(* CODESYS project 信号機_駅制御_柴山.project

Project tree, tasks and I/O mapping:
  Device : CODESYS Control Win V3 x64, 3S - Smart Software Solutions GmbH, version 3.5.11.40
    application Application
      libraries: Standard, * (System); File Access, 3.5.7.0 (3S - Smart Software Solutions GmbH); Network, 3.5.7.0 (3S - Smart Software Solutions GmbH)
      task MainTask (cyclic, interval 4 ms, priority 0) calls EtherCAT_Master.EtherCAT_Task [EtherCAT_Master.EtherCAT_Task], StationControlMain
      program StationControlMain [ST]
      function block OnOffDelay [ST]
      function block TrainDetection [ST]
      SignalControl/
        function block FourStateSignal [ST]
        function block FourStateSignalDecoder [ST]
        function block ThreeStateSignal [ST]
        function block ThreeStateSignalDecoder [ST]
        function block FourStateWarningSignalDecoder [ST]
      declarations NVL_StationControl
      global variables NVL_StationStatus
      global variables ControlLever
      function block SwitchControl [ST]
      function block SignalControl [ST]
      Encode/
        function block Encode_Status [ST]
        function EncodeSignalStatusOne [ST]
        function EncodeDetectionOne [ST]
        function EncodeSignalLockStatusOne [ST]
        function EncodeSwitchStatusOne [ST]
        function EncodeSwitchLockStatusOne [ST]
        function EncodeRouteStatusOne [ST]
      Decode/
        function DecodeSwitchLeverOne [ST]
        function block Decode_Levers [ST]
        function DecodeSignalLeverOne [ST]
      function block RouteControl [ST]
    EtherCAT_Master : EtherCAT Master, 3S - Smart Software Solutions GmbH, version 3.5.11.40
        settings: NetworkName = 'イーサネット'; NetworkName = "イーサネット"; SrcAddress1 = 60449; SrcAddress2 = 3851182877
      NX_ECC202 : NX-ECC202 EtherCAT coupler V1.2, OMRON Corporation, order no. NX-ECC202, version Revision=16#00010002
          settings: ModularDevice = True; Number of Outputs = 0; Number of Infos about Outputs = 0; MDP_InputOffsets = [0,0,0,0,272]; MDP_OutputOffsets = [0,0,32,64,0]; StationAlias = 0; Sync.Length = 12; Sync.Length = 38; FMMU.Length = 12; FMMU.Length = 38; Number of RxPDOs of the Slave = 3; Number of TxPDOs of the Slave = 4; DC sync0 cycletime = 4000; DC sync1 cycletime = 4000; Number of SDO = 1; RxTxPdo.NumberofExcludes = 0; RxTxPdo.NumberofEntries = 1; RxTxPdo.Index = 16#1600; RxTxPdo.Fixed = True; RxTxPdo.Mandatory = True; RxTxPdo.Virtual = False; RxTxPdo.Sm = 2; RxTxPdo.Su = 0; RxTxPdo.Name = 'Output Data Set 1'; RxTxPdo.DependOnSlot = True; RxTxPdo.DependOnSlotGroup = False; RxTxPdo.OverwrittenByModule = True; Output Bit 32 bits.Index = 16#7003; Output Bit 32 bits.SubIndex = 1; Output Bit 32 bits.Size = 32; Output Bit 32 bits.Offset = 0; Output Bit 32 bits.DependOnSlot = True; Output Bit 32 bits.DependOnSlotGroup = True; RxTxPdo.NumberofExcludes = 0; RxTxPdo.NumberofEntries = 1; RxTxPdo.Index = 16#1604; RxTxPdo.Fixed = True; RxTxPdo.Mandatory = True; RxTxPdo.Virtual = False; RxTxPdo.Sm = 2;
            RxTxPdo.Su = 0; RxTxPdo.Name = 'Output Data Set 1'; RxTxPdo.DependOnSlot = True; RxTxPdo.DependOnSlotGroup = False; RxTxPdo.OverwrittenByModule = True; Output Bit 32 bits.Index = 16#7023; Output Bit 32 bits.SubIndex = 1; Output Bit 32 bits.Size = 32; Output Bit 32 bits.Offset = 0; Output Bit 32 bits.DependOnSlot = True; Output Bit 32 bits.DependOnSlotGroup = True; RxTxPdo.NumberofExcludes = 0; RxTxPdo.NumberofEntries = 1; RxTxPdo.Index = 16#1608; RxTxPdo.Fixed = True; RxTxPdo.Mandatory = True; RxTxPdo.Virtual = False; RxTxPdo.Sm = 2; RxTxPdo.Su = 0; RxTxPdo.Name = 'Output Data Set 1'; RxTxPdo.DependOnSlot = True; RxTxPdo.DependOnSlotGroup = False; RxTxPdo.OverwrittenByModule = True; Output Bit 32 bits.Index = 16#7043; Output Bit 32 bits.SubIndex = 1; Output Bit 32 bits.Size = 32; Output Bit 32 bits.Offset = 0; Output Bit 32 bits.DependOnSlot = True; Output Bit 32 bits.DependOnSlotGroup = True; RxTxPdo.NumberofExcludes = 0; RxTxPdo.NumberofEntries = 2; RxTxPdo.Index = 16#1BF8; RxTxPdo.Fixed = False; RxTxPdo.Mandatory = False; RxTxPdo.Virtual = False; RxTxPdo.Sm = 3; RxTxPdo.Su = 3; RxTxPdo.Name = '505th transmit PDO Mapping'; RxTxPdo.DependOnSlot = False; RxTxPdo.DependOnSlotGroup = False;
            RxTxPdo.OverwrittenByModule = False; NX Unit Registration Status 125.Index = 16#3003; NX Unit Registration Status 125.SubIndex = 4; NX Unit Registration Status 125.Size = 128; NX Unit Registration Status 125.Offset = 0; NX Unit Registration Status 125.DependOnSlot = False; NX Unit Registration Status 125.DependOnSlotGroup = False; NX Unit I/O Data Active Status 125.Index = 16#3006; NX Unit I/O Data Active Status 125.SubIndex = 4; NX Unit I/O Data Active Status 125.Size = 128; NX Unit I/O Data Active Status 125.Offset = 0; NX Unit I/O Data Active Status 125.DependOnSlot = False; NX Unit I/O Data Active Status 125.DependOnSlotGroup = False; RxTxPdo.NumberofExcludes = 0; RxTxPdo.NumberofEntries = 1; RxTxPdo.Index = 16#1BFF; RxTxPdo.Fixed = True; RxTxPdo.Mandatory = False; RxTxPdo.Virtual = False; RxTxPdo.Sm = 3; RxTxPdo.Su = 3; RxTxPdo.Name = '512th transmit PDO Mapping'; RxTxPdo.DependOnSlot = False; RxTxPdo.DependOnSlotGroup = False; RxTxPdo.OverwrittenByModule = False; Sysmac Error Status.Index = 16#2002; Sysmac Error Status.SubIndex = 1; Sysmac Error Status.Size = 8; Sysmac Error Status.Offset = 0; Sysmac Error Status.DependOnSlot = False; Sysmac Error Status.DependOnSlotGroup = False; RxTxPdo.NumberofExcludes = 0; RxTxPdo.NumberofEntries = 1; RxTxPdo.Index = 16#1BF4; RxTxPdo.Fixed = True; RxTxPdo.Mandatory = False; RxTxPdo.Virtual = False; RxTxPdo.Sm = 3; RxTxPdo.Su = 3; RxTxPdo.Name = '501st transmit PDO Mapping';
            RxTxPdo.DependOnSlot = False; RxTxPdo.DependOnSlotGroup = False; RxTxPdo.OverwrittenByModule = False; Entry.Offset = 0; Entry.DependOnSlot = False; Entry.DependOnSlotGroup = False; RxTxPdo.NumberofExcludes = 0; RxTxPdo.NumberofEntries = 1; RxTxPdo.Index = 16#1A0C; RxTxPdo.Fixed = True; RxTxPdo.Mandatory = True; RxTxPdo.Virtual = False; RxTxPdo.Sm = 3; RxTxPdo.Su = 0; RxTxPdo.Name = 'Input Data Set  1'; RxTxPdo.DependOnSlot = True; RxTxPdo.DependOnSlotGroup = False; RxTxPdo.OverwrittenByModule = True; Input Bit 32 bits.Index = 16#6063; Input Bit 32 bits.SubIndex = 1; Input Bit 32 bits.Size = 32; Input Bit 32 bits.Offset = 0; Input Bit 32 bits.DependOnSlot = True; Input Bit 32 bits.DependOnSlotGroup = True; Output Bit 32 bits.Name = 'Output Bit 32 bits'; Output Bit 32 bits.DataType = 'UDINT'; Output Bit 32 bits.Default = ''; Output Bit 32 bits.Comment = ''; Output Bit 32 bits.Name = 'Output Bit 32 bits'; Output Bit 32 bits.DataType = 'UDINT'; Output Bit 32 bits.Default = ''; Output Bit 32 bits.Comment = ''; Output Bit 32 bits.Name = 'Output Bit 32 bits'; Output Bit 32 bits.DataType = 'UDINT'; Output Bit 32 bits.Default = ''; Output Bit 32 bits.Comment = ''; NX Unit Registration Status 125.Name = 'NX Unit Registration Status 125'; NX Unit Registration Status 125.DataType = 'ARRAY [0..15] OF BYTE'; NX Unit Registration Status 125.Default = ''; NX Unit Registration Status 125.Comment = '';
            NX Unit I/O Data Active Status 125.Name = 'NX Unit I/O Data Active Status 125'; NX Unit I/O Data Active Status 125.DataType = 'ARRAY [0..15] OF BYTE'; NX Unit I/O Data Active Status 125.Default = ''; NX Unit I/O Data Active Status 125.Comment = ''; Sysmac Error Status.Name = 'Sysmac Error Status'; Sysmac Error Status.DataType = 'USINT'; Sysmac Error Status.Default = ''; Sysmac Error Status.Comment = ''; Entry.Default = ''; Input Bit 32 bits.Name = 'Input Bit 32 bits'; Input Bit 32 bits.DataType = 'UDINT'; Input Bit 32 bits.Default = ''; Input Bit 32 bits.Comment = ''
          unmapped channels: NX Unit Registration Status 125, NX Unit I/O Data Active Status 125, Sysmac Error Status, 
        NX_OD6121_5 : General output, OMRON Corporation, order no. NX-OD6121-5, version 0
            settings: Number of Outputs = 1; Number of Infos about Outputs = 1; Output Bit 32 bits.Offset = 0; Output Bit 32 bits.DependOnSlot = True; Output Bit 32 bits.DependOnSlotGroup = True; Output Bit 32 bits.Default = ''
            unmapped channels: Output Bit 32 bits
        NX_ID6142_5_1 : General input, OMRON Corporation, order no. NX-ID6142-5, version 0
            settings: Number of Inputs = 1; Number of Infos about Inputs = 1; Input Bit 32 bits.Index = 16#6063; Input Bit 32 bits.SubIndex = 1; Input Bit 32 bits.Size = 32; Input Bit 32 bits.Offset = 0; Input Bit 32 bits.DependOnSlot = True; Input Bit 32 bits.DependOnSlotGroup = True; Input Bit 32 bits.Name = 'Input Bit 32 bits'; Input Bit 32 bits.DataType = 'UDINT'; Input Bit 32 bits.Default = ''; Input Bit 32 bits.Comment = ''
            unmapped channels: Input Bit 32 bits
        NX_OD6121_5_2 : General output, OMRON Corporation, order no. NX-OD6121-5, version 0
            settings: Number of Outputs = 1; Number of Infos about Outputs = 1; Output Bit 32 bits.Index = 16#7043; Output Bit 32 bits.SubIndex = 1; Output Bit 32 bits.Size = 32; Output Bit 32 bits.Offset = 0; Output Bit 32 bits.DependOnSlot = True; Output Bit 32 bits.DependOnSlotGroup = True; Output Bit 32 bits.Name = 'Output Bit 32 bits'; Output Bit 32 bits.DataType = 'UDINT'; Output Bit 32 bits.Default = ''; Output Bit 32 bits.Comment = ''
            unmapped channels: Output Bit 32 bits
        NX_OD6121_5_1 : General output, OMRON Corporation, order no. NX-OD6121-5, version 0
            settings: Number of Outputs = 1; Number of Infos about Outputs = 1; Output Bit 32 bits.Index = 16#7023; Output Bit 32 bits.SubIndex = 1; Output Bit 32 bits.Size = 32; Output Bit 32 bits.Offset = 0; Output Bit 32 bits.DependOnSlot = True; Output Bit 32 bits.DependOnSlotGroup = True; Output Bit 32 bits.Name = 'Output Bit 32 bits'; Output Bit 32 bits.DataType = 'UDINT'; Output Bit 32 bits.Default = ''; Output Bit 32 bits.Comment = ''
            unmapped channels: Output Bit 32 bits
  data type E_SIGNAL_STATUS
*)

// E_SIGNAL_STATUS
TYPE E_SIGNAL_STATUS :
(
	R_Stop, YY_Warnig, Y_Caution, YG_Slowdown, G_Go
);
END_TYPE

// Device/Application/NVL_StationControl
//このグローバル変数リストはネットワーク経由受信です。
//送信者: ファイル 'C:\Users\Tomonobu\Documents\home\CodesysProject\StationControl.gvl' からインポートされました
//プロトコル: UDP

{attribute 'qualified_only'}
VAR_GLOBAL
	singal_lever_status: ARRAY[0..15] OF UINT;
	switch_lever_nml: ARRAY[0..15] OF UINT;
	switch_lever_rev: ARRAY[0..15] OF UINT;
END_VAR

// Device/Application/NVL_StationStatus
{attribute 'qualified_only'}
VAR_GLOBAL
	signal_display: ARRAY[0..15] OF E_SIGNAL_STATUS;
	signal_satus: ARRAY[0..15] OF UINT;
	signal_locked: ARRAY[0..15] OF UINT;
	singal_reserve0: ARRAY[0..15] OF UINT;
	switch_status: ARRAY[0..15] OF UINT;
	switch_locked: ARRAY[0..15] OF UINT;
	switch_reserve0: ARRAY[0..15] OF UINT;
	section_status: ARRAY[0..15] OF UINT;
END_VAR

// Device/Application/ControlLever
{attribute 'qualified_only'}
VAR_GLOBAL
	Switch_31Nml: BOOL;
	Switch_21Nml: BOOL;
	Switch_31Rev: BOOL;
	Switch_21Rev: BOOL;
	Route_11Nml: BOOL;
	Route_11Rev: BOOL;
	Route_12Nml: BOOL;
	Route_12Rev: BOOL;
	Signal_2R: BOOL;
	Signal_3R: BOOL;
	Signal_4R: BOOL;
	Signal_5R: BOOL;
	Signal_2L: BOOL;
	Signal_3L: BOOL;
	Signal_4L: BOOL;
	Signal_5L: BOOL;
END_VAR

// Device/Application/StationControlMain
PROGRAM StationControlMain
VAR
	Detect_Sensor : TrainDetection; 
	Input_Decode  : Decode_Levers;
	Output_Encode : Encode_Status;
	abDetectInfo_All : ARRAY[0..15] OF BOOL;

	Signal_2R: SignalControl;
	Signal_3R: SignalControl;

	Signal_2L: SignalControl;
	Signal_3L: SignalControl;

	Route_11: RouteControl;
	Route_12: RouteControl;
	
	Switch_31: SwitchControl;
	Switch_21: SwitchControl;

	Signal_2L_Decode: FourStateWarningSignalDecoder;
	Signal_3L_Decode: ThreeStateSignalDecoder;
	Signal_2R_Decode: ThreeStateSignalDecoder;
 	Signal_3R_Decode: FourStateWarningSignalDecoder;
	
	// 在線検知
	bExist_31T: BOOL;
	bExist_21T: BOOL;
	bExist_2RT: BOOL;
	bExist_5RT: BOOL;
	
END_VAR

Input_Decode();
Output_Encode(sig_2R:=Signal_2R, sig_3R:=Signal_3R,
	          sig_2L:=Signal_2L, sig_3L:=Signal_3L,
			  swt_31:=Switch_31, swt_21:=Switch_21, 
			  route_11:=Route_11, route_12:=Route_12,
              abDetect:=abDetectInfo_All);
Detect_Sensor(abDetect => abDetectInfo_All);

// 在線検知信号
bExist_31T := abDetectInfo_All[0];
bExist_21T := abDetectInfo_All[1];
bExist_2RT := abDetectInfo_All[2];
bExist_5RT := abDetectInfo_All[3];

// 鎖錠信号
// 2L
IF NOT Switch_21.bStatusNormal THEN
	Signal_2L.bLockedNml := TRUE;
ELSE
	Signal_2L.bLockedNml := FALSE; 
END_IF
Signal_2L.bLockedRev := FALSE;

Signal_2L.bRouteAcquired := NOT Switch_31.bStatusNormal;

// 3L
IF Switch_31.bStatusNormal THEN
	Signal_3L.bLockedNml := TRUE;
ELSE
	SIgnal_3L.bLockedNml := FALSE;
END_IF

IF (Signal_2L.bLockActive AND NOT Signal_3L.bStatusNormal) THEN
	Signal_3L.bLockedRev := TRUE;
ELSE 
	Signal_3L.bLockedRev := FALSE;
END_IF

// 2R
IF Switch_21.bStatusNormal THEN
	Signal_2R.bLockedNml := TRUE;
ELSE
	Signal_2R.bLockedNml := FALSE;
END_IF

IF (Signal_3R.bLockActive AND NOT Signal_2R.bStatusNormal) THEN
	Signal_2R.bLockedRev := TRUE;
ELSE 
	Signal_2R.bLockedRev := FALSE;
END_IF

//5R
IF NOT Switch_31.bStatusNormal THEN
	Signal_3R.bLockedNml := TRUE;
ELSE
	Signal_3R.bLockedNml := FALSE;
END_IF
Signal_3R.bLockedRev := FALSE;

Signal_3R.bRouteAcquired := NOT Switch_21.bStatusNormal;

// 31
IF Signal_3R.bLockActive THEN
	Switch_31.bLockedNml := TRUE;
ELSE
	Switch_31.bLockedNml := FALSE;
END_IF

IF Signal_3L.bLockActive OR
	(Route_12.bLockActive AND NOT Switch_31.bStatusNormal) THEN
	Switch_31.bLockedRev := TRUE;
ELSE
	Switch_31.bLockedRev := FALSE;
END_IF

// 21
IF Signal_2L.bLockActive THEN
	Switch_21.bLockedNml := TRUE;
ELSE
	Switch_21.bLockedNml := FALSE;
END_IF

IF Signal_2R.bLockActive OR
	(Route_11.bLockActive AND NOT Switch_21.bStatusNormal) THEN
	Switch_21.bLockedRev := TRUE;
ELSE
	Switch_21.bLockedRev := FALSE;
END_IF

// 11
IF (Signal_3R.bLockActive AND NOT Route_11.bStatusNormal) THEN
	Route_11.bLockedRev := TRUE;
ELSE
	Route_11.bLockedRev := FALSE;
END_IF

// 12
IF (Signal_2L.bLockActive AND NOT Route_12.bStatusNormal) THEN
	Route_12.bLockedRev := TRUE;
ELSE
	Route_12.bLockedRev := FALSE;
END_IF


// 信号制御
Signal_2R.bDisplayControl := bExist_21T;
Signal_3R.bDisplayControl := bExist_31T OR bExist_2RT;
Signal_2L.bDisplayControl := bExist_21T OR bExist_5RT;
Signal_3L.bDisplayControl := bExist_31T;
Signal_2R.bRouteLock := bExist_21T;
Signal_3R.bRouteLock := bExist_31T;
Signal_2L.bRouteLock := bExist_21T;
Signal_3L.bRouteLock := bExist_31T;
Signal_2R.bRouteConfigured := NOT Switch_21.bStatusNormal;
Signal_3R.bRouteConfigured := Switch_31.bStatusNormal;
Signal_2L.bRouteConfigured := Switch_21.bStatusNormal;
Signal_3L.bRouteConfigured := NOT Switch_31.bStatusNormal;



// 信号機間の連動
Signal_2R.eNextSignalStatus := E_SIGNAL_STATUS.G_Go;
Signal_3R.eNextSignalStatus := Signal_2R.eSignalStatus;

Signal_2L.eNextSignalStatus := Signal_3L.eSignalStatus;
Signal_3L.eNextSignalStatus := E_SIGNAL_STATUS.G_Go;

// 信号機制御
Signal_2R(bLeverNormal := ControlLever.Signal_2R);
Signal_3R(bLeverNormal := ControlLever.Signal_3R, bConfig_DisplayWarning := TRUE);
Signal_2L(bLeverNormal := ControlLever.Signal_2L, bConfig_DisplayWarning := TRUE);
Signal_3L(bLeverNormal := ControlLever.Signal_3L);

// 開通てこ制御
IF NOT ControlLever.Signal_2R THEN
	Route_11.bConfigureRevReq := TRUE;
ELSE
	Route_11.bConfigureRevReq := FALSE;
END_IF

IF NOT ControlLever.Signal_3L THEN
	Route_12.bConfigureRevReq := TRUE;
ELSE
	Route_12.bConfigureRevReq := FALSE;	
END_IF
Route_11(bLeverNml := ControlLever.Route_11Nml, bLeverRev := ControlLever.Route_11Rev);
Route_12(bLeverNml := ControlLever.Route_12Nml, bLeverRev := ControlLever.Route_12Rev);

// 転轍機制御
IF NOT Route_11.bStatusNormal THEN
	Switch_21.bConfigureRevReq := TRUE;
ELSE
	Switch_21.bConfigureRevReq := FALSE;
END_IF

// 31
IF NOT Route_12.bStatusNormal THEN
	Switch_31.bConfigureRevReq := TRUE;
ELSE
	Switch_31.bConfigureRevReq := FALSE;
END_IF


Switch_31(bSwitchNml := ControlLever.Switch_31Nml,
			bSwitchRev := ControlLever.Switch_31Rev,
			bExistLock := bExist_31T);
Switch_21(bSwitchNml := ControlLever.Switch_21Nml,
			bSwitchRev := ControlLever.Switch_21Rev,
			bExistLock := bExist_21T);

// 信号機出力
Signal_2L_Decode(sSignalStatus:=Signal_2L.eSignalStatus);
Signal_3L_Decode(sSignalStatus:=Signal_3L.eSignalStatus);
Signal_2R_Decode(sSignalStatus:=Signal_2R.eSignalStatus);
Signal_3R_Decode(sSignalStatus:=Signal_3R.eSignalStatus);

%QX0.4 := Signal_2R_Decode.bGreen;
%QX0.5 := Signal_2R_Decode.bYellow;
%QX0.6 := Signal_2R_Decode.bRed;

%QX1.4 := Signal_3R_Decode.bYellow1;
%QX1.5 := Signal_3R_Decode.bRed;
%QX1.6 := Signal_3R_Decode.bGreen;
%QX1.7 := Signal_3R_Decode.bYellow2;

%QX2.0 := Signal_2L_Decode.bYellow1;
%QX2.1 := Signal_2L_Decode.bRed;
%QX2.2 := Signal_2L_Decode.bGreen;
%QX2.3 := Signal_2L_Decode.bYellow2;

%QX3.0 := Signal_3L_Decode.bGreen;
%QX3.1 := Signal_3L_Decode.bYellow;
%QX3.2 := Signal_3L_Decode.bRed;

// 転轍機出力
IF Switch_31.bStatusNormal THEN
	%QX4.0 := TRUE;
ELSE
	%QX4.0 := FALSE;
END_IF

IF Switch_21.bStatusNormal THEN
	%QX4.1 := TRUE;
ELSE
	%QX4.1 := FALSE;
END_IF

END_PROGRAM

// Device/Application/TrainDetection
FUNCTION_BLOCK TrainDetection
VAR_INPUT
END_VAR
VAR_OUTPUT
	abDetect: ARRAY[0..15] OF BOOL;
END_VAR
VAR
	DetectDelayExec: ARRAY[0..15] OF OnOffDelay;
	dwIdx: INT;
END_VAR

DetectDelayExec[0](bIN := %IX36.0);
DetectDelayExec[1](bIN := %IX36.1);
DetectDelayExec[2](bIN := %IX36.2);
DetectDelayExec[3](bIN := %IX36.3);
DetectDelayExec[4](bIN := %IX36.4);
FOR dwIdx:=0 TO 15 DO
	abDetect[dwIdx] := DetectDelayExec[dwIdx].bOUT;
END_FOR

END_FUNCTION_BLOCK

// Device/Application/OnOffDelay
FUNCTION_BLOCK OnOffDelay
VAR_INPUT
	bIN: BOOL;
END_VAR
VAR_OUTPUT
	bOUT: BOOL;
END_VAR
VAR
	OffDelayTimer: Standard.TOF;
	OnDelayTimer: Standard.TON;
	bPrevOutput: BOOL;
END_VAR

OffDelayTimer(IN:=bIN, PT:=T#0.5S);
OnDelayTimer(IN:=bIN, PT:=T#0.5S);
IF bPrevOutput THEN
	bOUT := OffDelayTimer.Q;
ELSE
	bOUT := OnDelayTimer.Q;	
END_IF
bPrevOutput := bOUT;

END_FUNCTION_BLOCK

// Device/Application/Decode/Decode_Levers
FUNCTION_BLOCK Decode_Levers
VAR_INPUT
END_VAR
VAR_OUTPUT
END_VAR
VAR
END_VAR

ControlLever.Signal_2R := DecodeSignalLeverOne(NVL_StationControl.singal_lever_status[0]);
ControlLever.Signal_3R := DecodeSignalLeverOne(NVL_StationControl.singal_lever_status[1]);
ControlLever.Signal_4R := DecodeSignalLeverOne(NVL_StationControl.singal_lever_status[2]);
ControlLever.Signal_5R := DecodeSignalLeverOne(NVL_StationControl.singal_lever_status[3]);
ControlLever.Signal_2L := DecodeSignalLeverOne(NVL_StationControl.singal_lever_status[4]);
ControlLever.Signal_3L := DecodeSignalLeverOne(NVL_StationControl.singal_lever_status[5]);
ControlLever.Signal_4L := DecodeSignalLeverOne(NVL_StationControl.singal_lever_status[6]);
ControlLever.Signal_5L := DecodeSignalLeverOne(NVL_StationControl.singal_lever_status[7]);

ControlLever.Switch_31Nml := DecodeSwitchLeverOne(NVL_StationControl.switch_lever_nml[0]);
ControlLever.Switch_21Nml := DecodeSwitchLeverOne(NVL_StationControl.switch_lever_nml[1]);
ControlLever.Route_11Nml := DecodeSwitchLeverOne(NVL_StationControl.switch_lever_nml[12]);
ControlLever.Route_12Nml := DecodeSwitchLeverOne(NVL_StationControl.switch_lever_nml[13]);

ControlLever.Switch_31Rev := DecodeSwitchLeverOne(NVL_StationControl.switch_lever_rev[0]);
ControlLever.Switch_21Rev := DecodeSwitchLeverOne(NVL_StationControl.switch_lever_rev[1]);
ControlLever.Route_11Rev := DecodeSwitchLeverOne(NVL_StationControl.switch_lever_rev[12]);
ControlLever.Route_12Rev := DecodeSwitchLeverOne(NVL_StationControl.switch_lever_rev[13]);

END_FUNCTION_BLOCK

// Device/Application/Decode/DecodeSignalLeverOne
FUNCTION DecodeSignalLeverOne : BOOL
VAR_INPUT
	Datalink_Val: UINT;
END_VAR
VAR
END_VAR

IF Datalink_Val = 1 THEN
	DecodeSignalLeverOne := FALSE;
ELSE
	DecodeSignalLeverOne := TRUE;	
END_IF

END_FUNCTION

// Device/Application/Decode/DecodeSwitchLeverOne
FUNCTION DecodeSwitchLeverOne : BOOL
VAR_INPUT
	Datalink_Val: UINT;
END_VAR
VAR
END_VAR

IF Datalink_Val = 1 THEN
	DecodeSwitchLeverOne := TRUE;
ELSE
	DecodeSwitchLeverOne := FALSE;	
END_IF

END_FUNCTION

// Device/Application/Encode/Encode_Status
FUNCTION_BLOCK Encode_Status
VAR_INPUT
	sig_2R: SignalControl;
	sig_3R: SignalControl;
	sig_4R: SignalControl;
	sig_5R: SignalControl;

	sig_2L: SignalControl;
	sig_3L: SignalControl;
	sig_4L: SignalControl;
	sig_5L: SignalControl;

	swt_31: SwitchControl;
	swt_21: SwitchControl;	
	
	route_11: RouteControl;
	route_12: RouteControl;
	
	abDetect: ARRAY[0..15] OF BOOL;
END_VAR
VAR_OUTPUT
END_VAR

NVL_StationStatus.signal_satus[0] := EncodeSignalStatusOne(sig_2R);
NVL_StationStatus.signal_satus[1] := EncodeSignalStatusOne(sig_3R);
NVL_StationStatus.signal_satus[2] := EncodeSignalStatusOne(sig_4R);
NVL_StationStatus.signal_satus[3] := EncodeSignalStatusOne(sig_5R);
NVL_StationStatus.signal_satus[4] := EncodeSignalStatusOne(sig_2L);
NVL_StationStatus.signal_satus[5] := EncodeSignalStatusOne(sig_3L);
NVL_StationStatus.signal_satus[6] := EncodeSignalStatusOne(sig_4L);
NVL_StationStatus.signal_satus[7] := EncodeSignalStatusOne(sig_5L);

NVL_StationStatus.switch_status[0] := EncodeSwitchStatusOne(swt_31);
NVL_StationStatus.switch_status[1] := EncodeSwitchStatusOne(swt_21);
NVL_StationStatus.switch_status[12] := EncodeRouteStatusOne(route_11);
NVL_StationStatus.switch_status[13] := EncodeRouteStatusOne(route_12);

NVL_StationStatus.section_status[0] := EncodeDetectionOne(abDetect[0]);
NVL_StationStatus.section_status[1] := EncodeDetectionOne(abDetect[1]);
NVL_StationStatus.section_status[2] := EncodeDetectionOne(abDetect[2]);
NVL_StationStatus.section_status[3] := EncodeDetectionOne(abDetect[3]);

NVL_StationStatus.signal_locked[0] := EncodeSignalLockStatusOne(sig_2R);
NVL_StationStatus.signal_locked[1] := EncodeSignalLockStatusOne(sig_3R);
NVL_StationStatus.signal_locked[2] := EncodeSignalLockStatusOne(sig_4R);
NVL_StationStatus.signal_locked[3] := EncodeSignalLockStatusOne(sig_5R);
NVL_StationStatus.signal_locked[4] := EncodeSignalLockStatusOne(sig_2L);
NVL_StationStatus.signal_locked[5] := EncodeSignalLockStatusOne(sig_3L);
NVL_StationStatus.signal_locked[6] := EncodeSignalLockStatusOne(sig_4L);
NVL_StationStatus.signal_locked[7] := EncodeSignalLockStatusOne(sig_5L);

NVL_StationStatus.switch_locked[0] := EncodeSwitchLockStatusOne(swt_31);
NVL_StationStatus.switch_locked[1] := EncodeSwitchLockStatusOne(swt_21);

END_FUNCTION_BLOCK

// Device/Application/Encode/EncodeSignalStatusOne
FUNCTION EncodeSignalStatusOne : UINT
VAR_INPUT
	signal: SignalControl;
END_VAR
VAR
END_VAR

IF signal.eSignalStatus = E_SIGNAL_STATUS.R_Stop THEN
	EncodeSignalStatusOne := 0;
ELSE
	EncodeSignalStatusOne := 1;
END_IF

END_FUNCTION

// Device/Application/SignalControl
FUNCTION_BLOCK SignalControl
VAR_INPUT
	bLeverNormal: BOOL;									// てこ状態
	bLockedNml: BOOL;
	bLockedRev: BOOL;
	bDisplayControl: BOOL;								// 現示制御
	bRouteLock: BOOL;									// 進路鎖錠
	bRouteConfigured: BOOL;								// 進路が構成されているか(接近鎖錠用)
	bRouteAcquired: BOOL;								// 過走防護の鎖錠ができているか
	eNextSignalStatus: E_SIGNAL_STATUS;
	bConfig_DisplayWarning: BOOL := FALSE;				// 警告現示が可能か
	bASRReq: BOOL;										// 接近鎖錠リレー動作
END_VAR
VAR_OUTPUT
	bStatusNormal: BOOL;
	eSignalStatus: E_SIGNAL_STATUS;
	bDisplayHold: BOOL;									// 保留現示
	bLockActive: BOOL;									// 鎖錠(接近鎖錠、進路鎖錠の論理和)
END_VAR
VAR
	bASR: BOOL;											// 接近鎖錠リレー
	ASRHoldTimer: Standard.TON;							// 保留鎖錠タイマ
	RouteLockHoldTimer: Standard.TOF;					// 進路鎖錠保留タイマ(接近鎖錠解除用)
END_VAR

// 状態制御
IF bLockedNml THEN
	// 定位に鎖錠されている
	bStatusNormal := TRUE;
ELSIF bLockedRev THEN	
	// 反位に鎖錠されている
	bStatusNormal := FALSE;
ELSIF bRouteLock THEN
	// 進路鎖錠
	bStatusNormal := FALSE;
ELSE
	// 鎖錠されていない
	IF NOT bLeverNormal THEN
		// 反位
		bStatusNormal := FALSE;
	ELSE
		// 定位
		bStatusNormal := TRUE;
	END_IF
END_IF

// 現示制御
IF (bStatusNormal 
	OR bDisplayHold) THEN
	eSignalStatus := E_SIGNAL_STATUS.R_Stop;
ELSE
	IF eNextSignalStatus = E_SIGNAL_STATUS.R_Stop THEN
		IF bRouteAcquired THEN
			// 過走防護の鎖錠あり
			eSignalStatus := E_SIGNAL_STATUS.Y_Caution;
		ELSE
			// 過走防護の鎖錠なし
			IF bConfig_DisplayWarning THEN
				eSignalStatus := E_SIGNAL_STATUS.YY_Warnig;
			ELSE
				eSignalStatus := E_SIGNAL_STATUS.R_Stop;
			END_IF
		END_IF
	ELSE
		eSignalStatus := E_SIGNAL_STATUS.G_Go;
	END_IF
END_IF

// 保留現示の制御
IF bStatusNormal THEN
	bDisplayHold := FALSE;
ELSE
 	IF bDisplayControl THEN
		bDisplayHold := TRUE;
	END_IF
END_IF

// 接近鎖錠制御
IF (eSignalStatus <> E_SIGNAL_STATUS.R_Stop)
	OR ((NOT bLeverNormal) AND bRouteConfigured) THEN
	bASR := TRUE;
END_IF

ASRHoldTimer(IN:=(bASR AND (eSignalStatus = E_SIGNAL_STATUS.R_Stop)), PT:=T#15S);
RouteLockHoldTimer(IN:=bRouteLock, PT:=T#30S);
IF bASR THEN
	IF (ASRHoldTimer.Q) THEN
		bASR := FALSE;
	END_IF
	IF (RouteLockHoldTimer.Q) THEN
		bASR := FALSE;
	END_IF
END_IF
IF bASR OR bRouteLock THEN
	bLockActive := TRUE;
ELSE
	bLockActive := FALSE;
END_IF

END_FUNCTION_BLOCK

// Device/Application/Encode/EncodeSwitchStatusOne
FUNCTION EncodeSwitchStatusOne : UINT
VAR_INPUT
	switch: SwitchControl;
END_VAR
VAR
END_VAR

IF switch.bStatusNormal THEN
	EncodeSwitchStatusOne := 0;
ELSE
	EncodeSwitchStatusOne := 1;
END_IF

END_FUNCTION

// Device/Application/SwitchControl
FUNCTION_BLOCK SwitchControl
VAR_INPUT
	bSwitchNml: BOOL;
	bSwitchRev: BOOL;
	bLockedNml: BOOL;
	bLockedRev: BOOL;
	bConfigureRevReq: BOOL;
	bExistLock: BOOL;			// てっさ鎖錠
END_VAR
VAR_OUTPUT
	bStatusNormal: BOOL;
END_VAR
VAR
END_VAR

IF NOT bExistLock THEN
	IF bSwitchNml THEN
		// 定位
		IF (NOT bLockedRev) THEN
			bStatusNormal := TRUE;
		ELSE
			bStatusNormal := FALSE;
		END_IF
	ELSIF bSwitchRev THEN
		// 反位
		IF (NOT bLockedNml) THEN
			bStatusNormal := FALSE;
		ELSE
			bStatusNormal := TRUE;
		END_IF
	ELSE
		IF ((NOT bLockedRev) AND (NOT bLockedNml)) THEN
			IF bConfigureRevReq THEN
				bStatusNormal := FALSE;
			ELSE
				bStatusNormal := TRUE;		
			END_IF
		END_IF
	END_IF
END_IF

END_FUNCTION_BLOCK

// Device/Application/Encode/EncodeRouteStatusOne
FUNCTION EncodeRouteStatusOne : UINT
VAR_INPUT
	route: RouteControl;
END_VAR
VAR
END_VAR

IF route.bStatusNormal THEN
	EncodeRouteStatusOne := 0;
ELSE
	EncodeRouteStatusOne := 1;
END_IF

END_FUNCTION

// Device/Application/RouteControl
FUNCTION_BLOCK RouteControl
// 開通てこ
VAR_INPUT
	bLeverNml: BOOL;									// てこ状態
	bLeverRev: BOOL;									// てこ状態
	bLockedNml: BOOL;
	bLockedRev: BOOL;	
	bConfigureNmlReq: BOOL;
	bConfigureRevReq: BOOL;
END_VAR
VAR_OUTPUT
	bLockActive: BOOL;
	bStatusNormal: BOOL;
END_VAR
VAR
END_VAR

IF bLockedNml THEN
	bStatusNormal := TRUE;
	bLockActive := FALSE;
ELSIF bLockedRev THEN
	bStatusNormal := FALSE;
	bLockActive := TRUE;
ELSE
	IF (bLeverRev OR bConfigureRevReq) THEN
		bStatusNormal := FALSE;
		bLockActive := TRUE;
	ELSE
		bStatusNormal := TRUE;
		bLockActive := FALSE;		 
	END_IF
END_IF

END_FUNCTION_BLOCK

// Device/Application/Encode/EncodeDetectionOne
FUNCTION EncodeDetectionOne : UINT
VAR_INPUT
	bIsDetect: BOOL;
END_VAR
VAR
END_VAR

IF bIsDetect THEN
	EncodeDetectionOne := 1;
ELSE
	EncodeDetectionOne := 0;
END_IF

END_FUNCTION

// Device/Application/Encode/EncodeSignalLockStatusOne
FUNCTION EncodeSignalLockStatusOne : UINT
VAR_INPUT
	signal: SignalControl;
END_VAR
VAR
END_VAR

IF(signal.bLockedNml OR signal.bLockedRev) THEN
	EncodeSignalLockStatusOne := 1;
ELSE
	EncodeSignalLockStatusOne := 0;
END_IF

END_FUNCTION

// Device/Application/Encode/EncodeSwitchLockStatusOne
FUNCTION EncodeSwitchLockStatusOne : UINT
VAR_INPUT
	switch: SwitchControl;
END_VAR
VAR
END_VAR

IF(switch.bLockedNml OR switch.bLockedRev) THEN
	EncodeSwitchLockStatusOne := 1;
ELSE
	EncodeSwitchLockStatusOne := 0;
END_IF

END_FUNCTION

// Device/Application/SignalControl/FourStateWarningSignalDecoder
FUNCTION_BLOCK FourStateWarningSignalDecoder
VAR_INPUT
	sSignalStatus: E_SIGNAL_STATUS;
END_VAR
VAR_OUTPUT
	bYellow1 : BOOL;
	bRed:     BOOL;
	bGreen:   BOOL;
	bYellow2: BOOL;
END_VAR
VAR
END_VAR

bYellow1 := FALSE;
bRed     := FALSE;
bGreen   := FALSE;
bYellow2 := FALSE;

IF sSignalStatus = R_Stop THEN
	bRed    := TRUE;
ELSIF sSignalStatus = Y_Caution THEN
	bYellow2 := TRUE;
ELSIF sSignalStatus = YY_Warnig THEN
	bYellow1 := TRUE;
	bYellow2 := TRUE;
ELSIF sSignalStatus = G_Go THEN
	bGreen  := TRUE;
END_IF

END_FUNCTION_BLOCK

// Device/Application/SignalControl/ThreeStateSignalDecoder
FUNCTION_BLOCK ThreeStateSignalDecoder
VAR_INPUT
	sSignalStatus: E_SIGNAL_STATUS;
END_VAR
VAR_OUTPUT
	bRed:     BOOL;
	bYellow : BOOL;
	bGreen:   BOOL;
END_VAR
VAR
END_VAR

bYellow  := FALSE;
bRed     := FALSE;
bGreen   := FALSE;


IF sSignalStatus = R_Stop THEN
	bRed    := TRUE;
ELSIF sSignalStatus = Y_Caution THEN
	bYellow := TRUE;
ELSIF sSignalStatus = G_Go THEN
	bGreen  := TRUE;
END_IF

END_FUNCTION_BLOCK

// Device/Application/SignalControl/FourStateSignal
FUNCTION_BLOCK FourStateSignal
VAR_INPUT
	bExist: BOOL;
	sNextSignalStatus: E_SIGNAL_STATUS;
END_VAR
VAR_OUTPUT
	sSignalStatus: E_SIGNAL_STATUS;
END_VAR
VAR
END_VAR

IF  bExist THEN
	sSignalStatus := R_Stop;
ELSE
	CASE sNextSignalStatus OF
	R_Stop : sSignalStatus := Y_Caution;
	YY_Warnig : sSignalStatus := Y_Caution;
	Y_Caution : sSignalStatus := YG_Slowdown;
	ELSE
		sSignalStatus := G_Go;
	END_CASE
END_IF

END_FUNCTION_BLOCK

// Device/Application/SignalControl/FourStateSignalDecoder
FUNCTION_BLOCK FourStateSignalDecoder
VAR_INPUT
	sSignalStatus: E_SIGNAL_STATUS;
END_VAR
VAR_OUTPUT
	bDummy:   BOOL;
	bYellow1: BOOL;
	bRed:     BOOL;
	bYellow2:  BOOL;
	bGreen:   BOOL;
END_VAR
VAR
END_VAR

bYellow1 := FALSE;
bRed     := FALSE;
bYellow2 := FALSE;
bGreen   := FALSE;


IF sSignalStatus = R_Stop THEN
	bRed := TRUE;
ELSIF sSignalStatus = Y_Caution THEN
	bYellow2 := TRUE;
ELSIF sSignalStatus = YG_Slowdown THEN
	bYellow1 := TRUE;
	bGreen := TRUE;
ELSIF sSignalStatus = G_Go THEN
	bGreen := TRUE;
END_IF

END_FUNCTION_BLOCK

// Device/Application/SignalControl/ThreeStateSignal
FUNCTION_BLOCK ThreeStateSignal
VAR_INPUT
	bExist: BOOL;
	sNextSignalStatus: E_SIGNAL_STATUS;
END_VAR
VAR_OUTPUT
	sSignalStatus: E_SIGNAL_STATUS;
END_VAR
VAR
END_VAR

IF  bExist THEN
	sSignalStatus := R_Stop;
ELSE
	CASE sNextSignalStatus OF
	R_Stop    : sSignalStatus := Y_Caution;
	YY_Warnig : sSignalStatus := Y_Caution;
	ELSE
		sSignalStatus := G_Go;
	END_CASE
END_IF

END_FUNCTION_BLOCK
